PROGRAM POU_Clamp
VAR
END_VAR

END_PROGRAM

(* stored: Version 1.1.0.1, ProductVersion 3.1.4024.12
   POU POU_Clamp: Id {1f4ba244-669d-4445-be61-dc452ae93b0d}, SpecialFunc None *)
